Fanuc TP program (LS listing): mv_to_place.ls

/PROG  MV_TO_PLACE
/ATTR
DEFAULT_GROUP	= 1,*,*,*,*;
/MN
 : CALL MV_RETREAT ;
 :  ;
 : UFRAME_NUM=${UF_PLACE} ;
 : UTOOL_NUM=${UT_PLACE} ;
 : J PR{PLACE_PERCH} ${PERCH_SPEED}% CNT100 ;
/POS
/END
